{attribute addProperty BoxType "EK1122-0000-0018"}
{attribute addProperty Id "Beckhoff_ELM37xxsub_EK1100EK1100_179A0949162"}
{attribute addProperty CRC "4214442396"}
{attribute addProperty SizeInBites "16"}
{attribute addProperty SizeInBytes "2"}
TYPE Beckhoff_ELM37xxEK1122_FB33499C EXTENDS EK1122_179A0949 :
STRUCT
	{attribute addProperty Name "Beckhoff_ELM37xxsub_EK1100"}
	Beckhoff_ELM37xxsub_EK1100 : EK1100_179A0949;
END_STRUCT
END_TYPE

(* stored: Version 1.2.0.0, ProductVersion 3.1.4024.9
   DUT Beckhoff_ELM37xxEK1122_FB33499C: Id {9c13aa04-fbe8-499c-9bc8-34d06dba4d56} *)
